FUNCTION_BLOCK DropSinkService (* Message Exchange example (slide 47): DSServ - service-oriented drop sink, acknowledges every drop request *)
  (* Standard: 61499-2; Description: Copyright (c) 2026 Meisterschulen am Ostbahnhof This program and the accompanying materials are made available under the terms of the Eclipse Public License 2.0 which is available at https://www.eclipse.org/legal/epl-2.0/ SPDX-License-Identifier: EPL-2.0 *)
  (* Version 1.0, 2026-09-03, Franz Höpfinger, Meisterschulen am Ostbahnhof, SoA implementation in function blocks (IEC 61499 primer course, Module 6, Valeriy Vyatkin, slide 47), DSServ role: uses EVENT_HS_ACK_WSTRING (REQ/CNF only, no IND/RSP needed - the sink never sends unsolicited notifications) *)
  PACKAGE Meins::DesingPatterns::HandshakePattern;
  IMPORT Meins::DesingPatterns::HandshakePattern::const::MessageExchangeConst;
  (* Documentation:
  Service-oriented drop sink (DSServ in the "SoA implementation in function blocks" diagram, IEC 61499 primer course, Module 6, Valeriy Vyatkin, slide 47) - one of the four function blocks in the CylH message-exchange example (slides 42-46 for the message sequence chart this reconstructs).
   Uses EVENT_HS_ACK_WSTRING as a Socket: every REQ (expected payload MessageExchangeConst::REQ_DROP, i.e. "drop") is unconditionally acknowledged with CNF carrying MessageExchangeConst::RSP_ACK ("ack") - matching the MSC's REQ,"drop" / RSP,"ack" exchange between CYL and DS. No IND/RSP needed: the sink never sends an unsolicited notification.
   See HandshakePattern.md in this folder, section "Die Quelle der 'push,100'-Notation", for the full write-up and the other three function blocks of this example (WorkpieceSensor, CylinderOrchestrator, CylinderService).
  *)
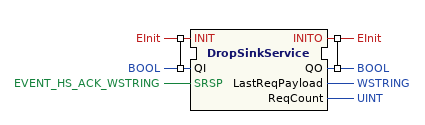
  EVENT_INPUT
    INIT : EInit WITH QI; (* Initialization Request *)
  END_EVENT
  EVENT_OUTPUT
    INITO : EInit WITH QO; (* Initialization Confirm *)
  END_EVENT
  VAR_INPUT
    QI : BOOL; (* Input event qualifier *)
  END_VAR
  VAR_OUTPUT
    QO : BOOL; (* Output event qualifier *)
    LastReqPayload : WSTRING; (* Payload of the last received REQ (expected: MessageExchangeConst::REQ_DROP) *)
    ReqCount : UINT; (* Number of drop REQ received (demo counter) *)
  END_VAR
  SOCKETS
    SRSP : adapter::types::bidirectional::Handshake::EVENT_HS_ACK_WSTRING; (* Service socket: receives REQ (+REQD), answers with CNF (+CNFD) *)
  END_SOCKETS
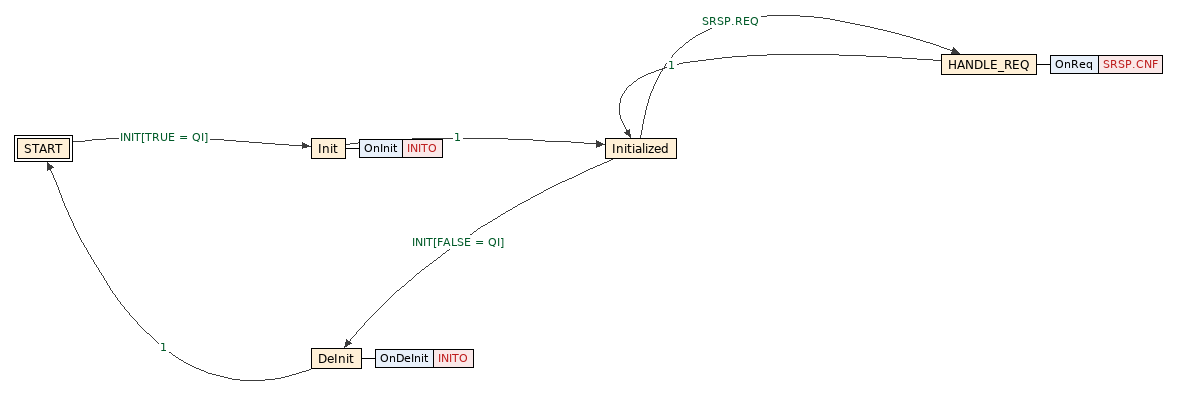
  EC_STATES
    START; (* Uninitialized *)
    Init : OnInit -> INITO; (* Initialization *)
    Initialized; (* Idle, ready to react *)
    DeInit : OnDeInit -> INITO; (* De-initialization *)
    HANDLE_REQ : OnReq -> SRSP.CNF; (* Read REQD, acknowledge every drop with RSP_ACK *)
  END_STATES
  EC_TRANSITIONS
    START TO Init := INIT[TRUE = QI];
    Init TO Initialized := 1;
    Initialized TO DeInit := INIT[FALSE = QI];
    DeInit TO START := 1;
    Initialized TO HANDLE_REQ := SRSP.REQ;
    HANDLE_REQ TO Initialized := 1;
  END_TRANSITIONS
  ALGORITHM OnInit IN ST: (* Reset demo counters *)
LastReqPayload := "";
ReqCount := 0;
QO := QI;
  END_ALGORITHM
  ALGORITHM OnDeInit IN ST: (* De-initialize *)
QO := FALSE;
  END_ALGORITHM
  ALGORITHM OnReq IN ST: (* Read REQD, count it, always answer with the fixed ack payload *)
LastReqPayload := SRSP.REQD;
ReqCount := ReqCount + 1;
SRSP.CNFD := MessageExchangeConst::RSP_ACK;
  END_ALGORITHM
END_FUNCTION_BLOCK
